///Error history type
TYPE T_ErrorHistory : ARRAY[GVL_ObjectSetup.cErrorHistMin..GVL_ObjectSetup.cErrorHistMax] OF DWORD; END_TYPE

(* stored: Version 1.1.0.1, ProductVersion 3.1.4019.2
   DUT T_ErrorHistory: Id {43b6c0da-4363-4a91-9d60-bb17a15cdeb9} *)
